//==================================================================================================
//								RJM Maszyny sp. z o.o.
//									04.02.2022
//	Obsługa elektrozaworu 5/3 zapowietrzony w pozycji środkowej
// 	v1.0	|| TC v 3.1.4024.22		|| - pierwsza wersja
//==================================================================================================
FUNCTION_BLOCK FB_Elektrozawor_5na3_Zapowietrzony IMPLEMENTS I_Elektrozawor_5na
VAR
	fbCewkaA								: FB_ElektrozaworCewka;
	fbCewkaB								: FB_ElektrozaworCewka;
END_VAR

//==================================================================================================
//								RJM Maszyny sp. z o.o.
//									04.02.2022
//	Włączenie cewki - wyjscie 2
// 	v1.0	|| TC v 3.1.4024.22		|| - pierwsza wersja
//==================================================================================================
METHOD WlaczWyjscie2 : BOOL
VAR_INPUT
END_VAR
fbCewkaA.Wylacz ();
END_METHOD

//==================================================================================================
//								RJM Maszyny sp. z o.o.
//									04.02.2022
//	Włączenie cewki - wyjscie 4
// 	v1.0	|| TC v 3.1.4024.22		|| - pierwsza wersja
//==================================================================================================
METHOD WlaczWyjscie4 : BOOL
VAR_INPUT
END_VAR
fbCewkaB.Wylacz ();
END_METHOD

//==================================================================================================
//								RJM Maszyny sp. z o.o.
//									04.02.2022
//	Wyłączenie cewki - wyjscie 2
// 	v1.0	|| TC v 3.1.4024.22		|| - pierwsza wersja
//==================================================================================================
METHOD WylaczWyjscie2 : BOOL
VAR_INPUT
END_VAR
fbCewkaA.Wlacz ();
END_METHOD

//==================================================================================================
//								RJM Maszyny sp. z o.o.
//									04.02.2022
//	Wyłączenie cewki - wyjscie 4
// 	v1.0	|| TC v 3.1.4024.22		|| - pierwsza wersja
//==================================================================================================
METHOD WylaczWyjscie4 : BOOL
VAR_INPUT
END_VAR
fbCewkaB.Wlacz ();
END_METHOD

END_FUNCTION_BLOCK

(* stored: Version 1.1.0.1, ProductVersion 3.1.4024.11
   POU FB_Elektrozawor_5na3_Zapowietrzony: Id {3442b49e-fb5a-45e5-929b-5abafebce8b5}, SpecialFunc None
   Method WlaczWyjscie2: Id {a80d863d-1ed3-44b0-bd88-83c724491f2e}
   Method WlaczWyjscie4: Id {61e05419-a3ea-4866-9827-4c84e80e73aa}
   Method WylaczWyjscie2: Id {d13d58dc-ad63-49ea-81e8-18aa1523c24b}
   Method WylaczWyjscie4: Id {652189a6-d336-4f57-905f-7726f3aaa32e} *)
